PROGRAM InitSIEMENSInput
VAR
	fbActPowerRQ: fbDwordToReal;
	fbReactPowerRQ: fbDwordToReal;
	fbGenActPower: fbDwordToReal;
	fbGenReactPower: fbDwordToReal;
	fbGenFreq: fbWordToReal;
	fbGenLineVoltage: fbWordToReal;
	fbMinSOCCustomer: fbWordToReal;
	fbMaxSOCCustomer: fbWordToReal;
	fbInvCurrentRampRate: fbDWordToReal;
	fbFreqDroop: fbWordToReal;
	fbVoltageDroop: fbWordToReal;
	fbInvNomVolt: fbWordToReal;
	fbInvNomFreq: fbWordToReal;
	fbCurrentLimMax: fbWordToReal;
	fbCurrentLimMin: fbWordToReal;
	fbGVoltageA		: fbWordToReal;
	fbGVoltageB		: fbWordToReal;
	fbGVoltageC		: fbWordToReal;
	fbGVoltageAB	: fbWordToReal;
	fbGVoltageBC	: fbWordToReal;
	fbGVoltageCA	: fbWordToReal;
	fbGCurrentL1	: fbWordToReal;
	fbGCurrentL2	: fbWordToReal;
	fbGCurrentL3	: fbWordToReal;
END_VAR

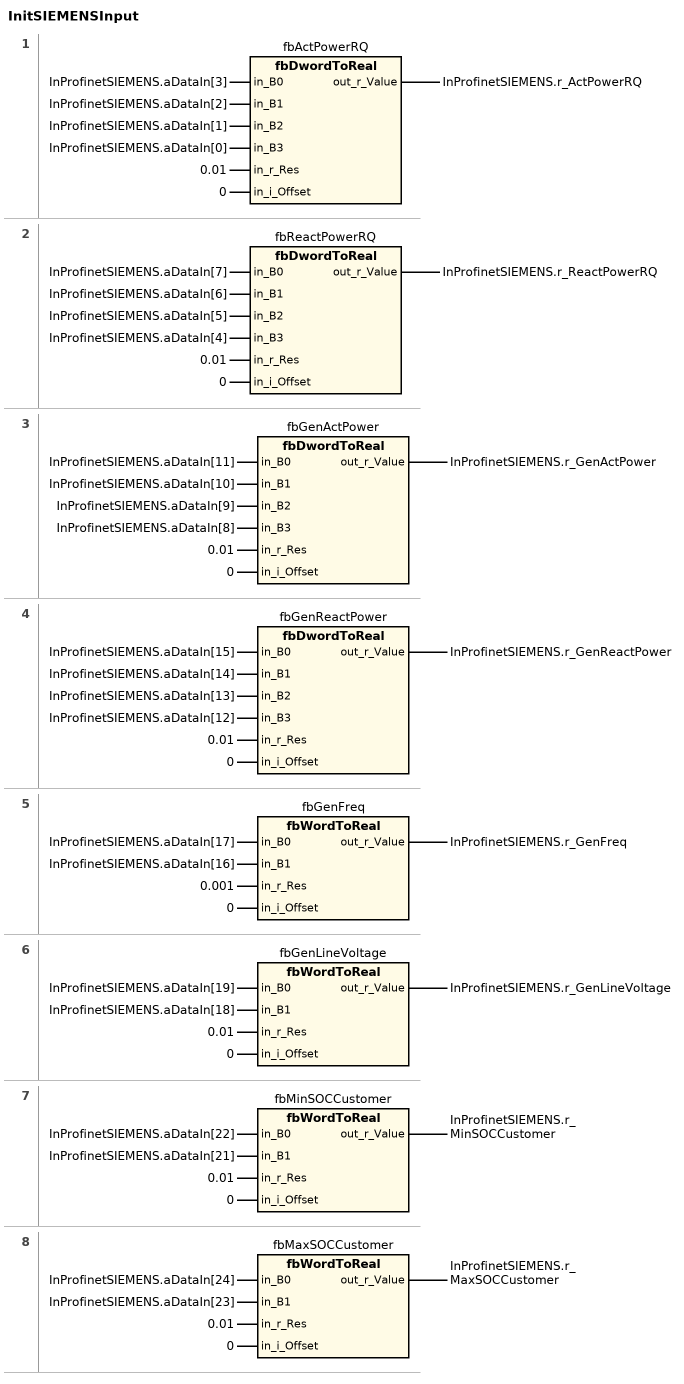
// NETWORK 1
fbActPowerRQ(
    in_B0 := InProfinetSIEMENS.aDataIn[3],
    in_B1 := InProfinetSIEMENS.aDataIn[2],
    in_B2 := InProfinetSIEMENS.aDataIn[1],
    in_B3 := InProfinetSIEMENS.aDataIn[0],
    in_r_Res := 0.01,
    in_i_Offset := 0); // fbDwordToReal
InProfinetSIEMENS.r_ActPowerRQ := fbActPowerRQ.out_r_Value;

// NETWORK 2
fbReactPowerRQ(
    in_B0 := InProfinetSIEMENS.aDataIn[7],
    in_B1 := InProfinetSIEMENS.aDataIn[6],
    in_B2 := InProfinetSIEMENS.aDataIn[5],
    in_B3 := InProfinetSIEMENS.aDataIn[4],
    in_r_Res := 0.01,
    in_i_Offset := 0); // fbDwordToReal
InProfinetSIEMENS.r_ReactPowerRQ := fbReactPowerRQ.out_r_Value;

// NETWORK 3
fbGenActPower(
    in_B0 := InProfinetSIEMENS.aDataIn[11],
    in_B1 := InProfinetSIEMENS.aDataIn[10],
    in_B2 := InProfinetSIEMENS.aDataIn[9],
    in_B3 := InProfinetSIEMENS.aDataIn[8],
    in_r_Res := 0.01,
    in_i_Offset := 0); // fbDwordToReal
InProfinetSIEMENS.r_GenActPower := fbGenActPower.out_r_Value;

// NETWORK 4
fbGenReactPower(
    in_B0 := InProfinetSIEMENS.aDataIn[15],
    in_B1 := InProfinetSIEMENS.aDataIn[14],
    in_B2 := InProfinetSIEMENS.aDataIn[13],
    in_B3 := InProfinetSIEMENS.aDataIn[12],
    in_r_Res := 0.01,
    in_i_Offset := 0); // fbDwordToReal
InProfinetSIEMENS.r_GenReactPower := fbGenReactPower.out_r_Value;

// NETWORK 5
fbGenFreq(
    in_B0 := InProfinetSIEMENS.aDataIn[17],
    in_B1 := InProfinetSIEMENS.aDataIn[16],
    in_r_Res := 0.001,
    in_i_Offset := 0); // fbWordToReal
InProfinetSIEMENS.r_GenFreq := fbGenFreq.out_r_Value;

// NETWORK 6
fbGenLineVoltage(
    in_B0 := InProfinetSIEMENS.aDataIn[19],
    in_B1 := InProfinetSIEMENS.aDataIn[18],
    in_r_Res := 0.01,
    in_i_Offset := 0); // fbWordToReal
InProfinetSIEMENS.r_GenLineVoltage := fbGenLineVoltage.out_r_Value;

// NETWORK 7
fbMinSOCCustomer(
    in_B0 := InProfinetSIEMENS.aDataIn[22],
    in_B1 := InProfinetSIEMENS.aDataIn[21],
    in_r_Res := 0.01,
    in_i_Offset := 0); // fbWordToReal
InProfinetSIEMENS.r_MinSOCCustomer := fbMinSOCCustomer.out_r_Value;

// NETWORK 8
fbMaxSOCCustomer(
    in_B0 := InProfinetSIEMENS.aDataIn[24],
    in_B1 := InProfinetSIEMENS.aDataIn[23],
    in_r_Res := 0.01,
    in_i_Offset := 0); // fbWordToReal
InProfinetSIEMENS.r_MaxSOCCustomer := fbMaxSOCCustomer.out_r_Value;

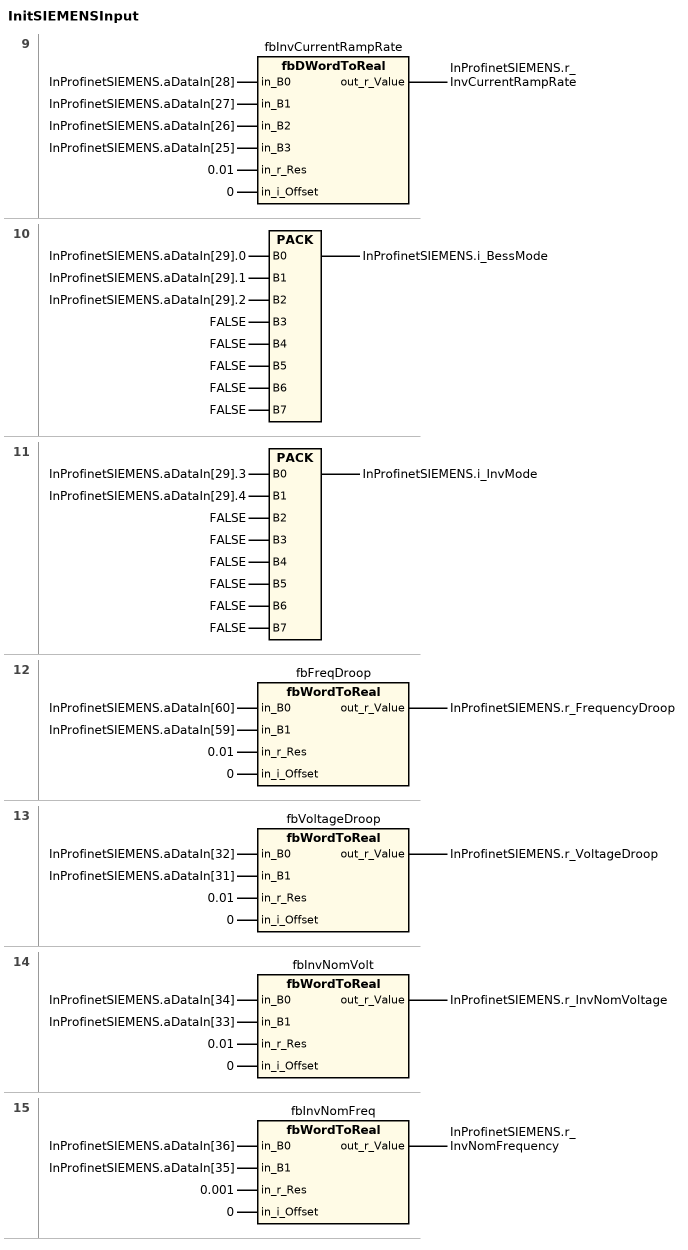
// NETWORK 9
fbInvCurrentRampRate(
    in_B0 := InProfinetSIEMENS.aDataIn[28],
    in_B1 := InProfinetSIEMENS.aDataIn[27],
    in_B2 := InProfinetSIEMENS.aDataIn[26],
    in_B3 := InProfinetSIEMENS.aDataIn[25],
    in_r_Res := 0.01,
    in_i_Offset := 0); // fbDWordToReal
InProfinetSIEMENS.r_InvCurrentRampRate := fbInvCurrentRampRate.out_r_Value;

// NETWORK 10
InProfinetSIEMENS.i_BessMode := PACK(B0 := InProfinetSIEMENS.aDataIn[29].0, B1 := InProfinetSIEMENS.aDataIn[29].1, B2 := InProfinetSIEMENS.aDataIn[29].2, B3 := FALSE, B4 := FALSE, B5 := FALSE, B6 := FALSE, B7 := FALSE);

// NETWORK 11
InProfinetSIEMENS.i_InvMode := PACK(B0 := InProfinetSIEMENS.aDataIn[29].3, B1 := InProfinetSIEMENS.aDataIn[29].4, B2 := FALSE, B3 := FALSE, B4 := FALSE, B5 := FALSE, B6 := FALSE, B7 := FALSE);

// NETWORK 12
fbFreqDroop(
    in_B0 := InProfinetSIEMENS.aDataIn[60],
    in_B1 := InProfinetSIEMENS.aDataIn[59],
    in_r_Res := 0.01,
    in_i_Offset := 0); // fbWordToReal
InProfinetSIEMENS.r_FrequencyDroop := fbFreqDroop.out_r_Value;

// NETWORK 13
fbVoltageDroop(
    in_B0 := InProfinetSIEMENS.aDataIn[32],
    in_B1 := InProfinetSIEMENS.aDataIn[31],
    in_r_Res := 0.01,
    in_i_Offset := 0); // fbWordToReal
InProfinetSIEMENS.r_VoltageDroop := fbVoltageDroop.out_r_Value;

// NETWORK 14
fbInvNomVolt(
    in_B0 := InProfinetSIEMENS.aDataIn[34],
    in_B1 := InProfinetSIEMENS.aDataIn[33],
    in_r_Res := 0.01,
    in_i_Offset := 0); // fbWordToReal
InProfinetSIEMENS.r_InvNomVoltage := fbInvNomVolt.out_r_Value;

// NETWORK 15
fbInvNomFreq(
    in_B0 := InProfinetSIEMENS.aDataIn[36],
    in_B1 := InProfinetSIEMENS.aDataIn[35],
    in_r_Res := 0.001,
    in_i_Offset := 0); // fbWordToReal
InProfinetSIEMENS.r_InvNomFrequency := fbInvNomFreq.out_r_Value;

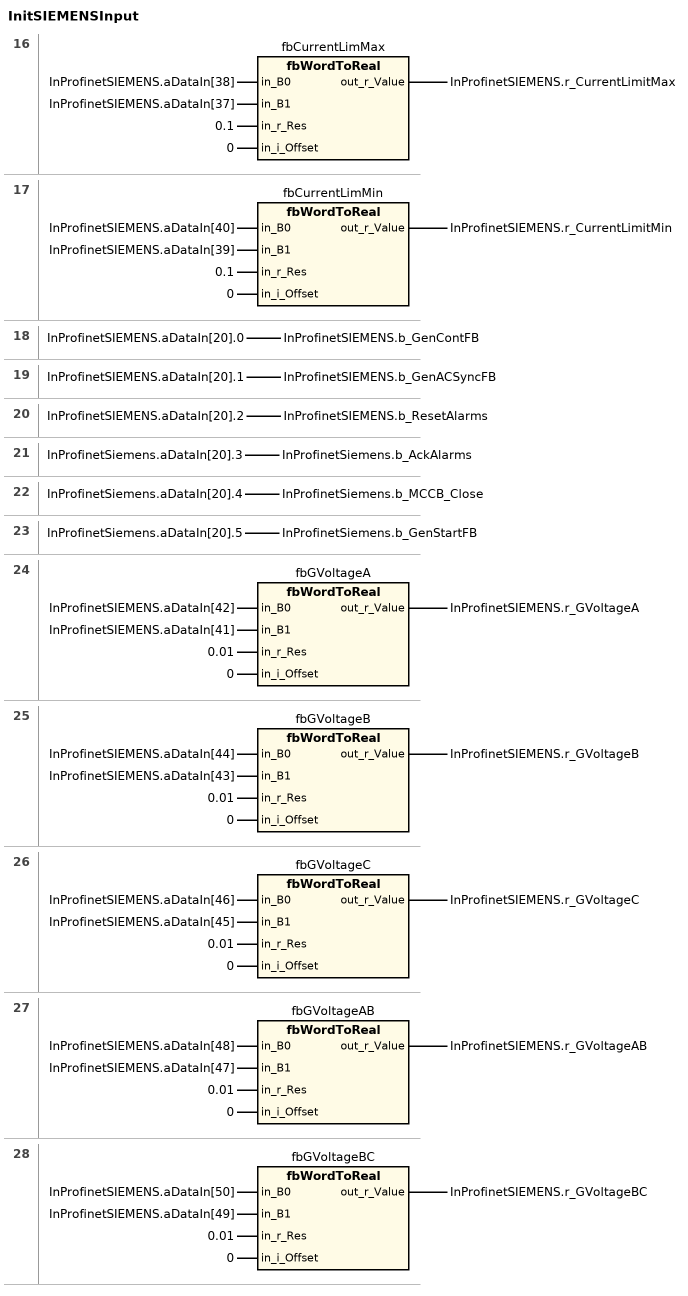
// NETWORK 16
fbCurrentLimMax(
    in_B0 := InProfinetSIEMENS.aDataIn[38],
    in_B1 := InProfinetSIEMENS.aDataIn[37],
    in_r_Res := 0.1,
    in_i_Offset := 0); // fbWordToReal
InProfinetSIEMENS.r_CurrentLimitMax := fbCurrentLimMax.out_r_Value;

// NETWORK 17
fbCurrentLimMin(
    in_B0 := InProfinetSIEMENS.aDataIn[40],
    in_B1 := InProfinetSIEMENS.aDataIn[39],
    in_r_Res := 0.1,
    in_i_Offset := 0); // fbWordToReal
InProfinetSIEMENS.r_CurrentLimitMin := fbCurrentLimMin.out_r_Value;

// NETWORK 18
InProfinetSIEMENS.b_GenContFB := InProfinetSIEMENS.aDataIn[20].0;

// NETWORK 19
InProfinetSIEMENS.b_GenACSyncFB := InProfinetSIEMENS.aDataIn[20].1;

// NETWORK 20
InProfinetSIEMENS.b_ResetAlarms := InProfinetSIEMENS.aDataIn[20].2;

// NETWORK 21
InProfinetSiemens.b_AckAlarms := InProfinetSiemens.aDataIn[20].3;

// NETWORK 22
InProfinetSiemens.b_MCCB_Close := InProfinetSiemens.aDataIn[20].4;

// NETWORK 23
InProfinetSiemens.b_GenStartFB := InProfinetSiemens.aDataIn[20].5;

// NETWORK 24
fbGVoltageA(
    in_B0 := InProfinetSIEMENS.aDataIn[42],
    in_B1 := InProfinetSIEMENS.aDataIn[41],
    in_r_Res := 0.01,
    in_i_Offset := 0); // fbWordToReal
InProfinetSIEMENS.r_GVoltageA := fbGVoltageA.out_r_Value;

// NETWORK 25
fbGVoltageB(
    in_B0 := InProfinetSIEMENS.aDataIn[44],
    in_B1 := InProfinetSIEMENS.aDataIn[43],
    in_r_Res := 0.01,
    in_i_Offset := 0); // fbWordToReal
InProfinetSIEMENS.r_GVoltageB := fbGVoltageB.out_r_Value;

// NETWORK 26
fbGVoltageC(
    in_B0 := InProfinetSIEMENS.aDataIn[46],
    in_B1 := InProfinetSIEMENS.aDataIn[45],
    in_r_Res := 0.01,
    in_i_Offset := 0); // fbWordToReal
InProfinetSIEMENS.r_GVoltageC := fbGVoltageC.out_r_Value;

// NETWORK 27
fbGVoltageAB(
    in_B0 := InProfinetSIEMENS.aDataIn[48],
    in_B1 := InProfinetSIEMENS.aDataIn[47],
    in_r_Res := 0.01,
    in_i_Offset := 0); // fbWordToReal
InProfinetSIEMENS.r_GVoltageAB := fbGVoltageAB.out_r_Value;

// NETWORK 28
fbGVoltageBC(
    in_B0 := InProfinetSIEMENS.aDataIn[50],
    in_B1 := InProfinetSIEMENS.aDataIn[49],
    in_r_Res := 0.01,
    in_i_Offset := 0); // fbWordToReal
InProfinetSIEMENS.r_GVoltageBC := fbGVoltageBC.out_r_Value;

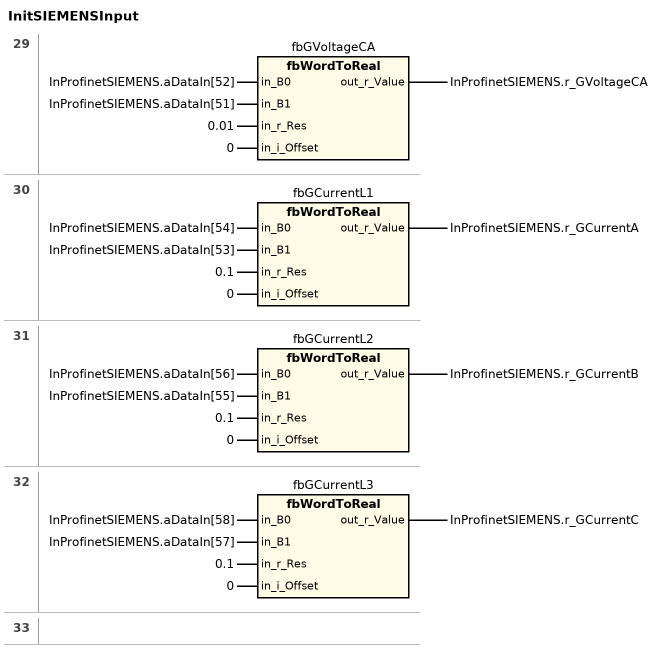
// NETWORK 29
fbGVoltageCA(
    in_B0 := InProfinetSIEMENS.aDataIn[52],
    in_B1 := InProfinetSIEMENS.aDataIn[51],
    in_r_Res := 0.01,
    in_i_Offset := 0); // fbWordToReal
InProfinetSIEMENS.r_GVoltageCA := fbGVoltageCA.out_r_Value;

// NETWORK 30
fbGCurrentL1(
    in_B0 := InProfinetSIEMENS.aDataIn[54],
    in_B1 := InProfinetSIEMENS.aDataIn[53],
    in_r_Res := 0.1,
    in_i_Offset := 0); // fbWordToReal
InProfinetSIEMENS.r_GCurrentA := fbGCurrentL1.out_r_Value;

// NETWORK 31
fbGCurrentL2(
    in_B0 := InProfinetSIEMENS.aDataIn[56],
    in_B1 := InProfinetSIEMENS.aDataIn[55],
    in_r_Res := 0.1,
    in_i_Offset := 0); // fbWordToReal
InProfinetSIEMENS.r_GCurrentB := fbGCurrentL2.out_r_Value;

// NETWORK 32
fbGCurrentL3(
    in_B0 := InProfinetSIEMENS.aDataIn[58],
    in_B1 := InProfinetSIEMENS.aDataIn[57],
    in_r_Res := 0.1,
    in_i_Offset := 0); // fbWordToReal
InProfinetSIEMENS.r_GCurrentC := fbGCurrentL3.out_r_Value;

// NETWORK 33

END_PROGRAM

(* stored: Version 1.1.0.1, ProductVersion 3.1.4024.12
   POU InitSIEMENSInput: Id {695d4762-9390-41f7-89b1-6b6446ab776f}, SpecialFunc None *)
